TEXTLIST E_ComponentTypes
  0 = 'NA'
  10 = 'Cylinder'
  11 = 'Axis'
  20 = 'EstopButton'
  21 = 'EstopBumper'
  22 = 'Pushbutton'
  23 = 'Switch'
  30 = 'SafeIO'
  31 = 'Rio_Box'
  32 = 'Rio_Slot'
  33 = 'Encoder'
  34 = 'DiSensor'
  40 = 'ServoDrive'
  50 = 'HMI'
  51 = 'RemoteOS'
  52 = 'RemoteDB'
  60 = 'Assembly'
  61 = 'SubAssembly'
  100 = 'MainProgram'
  101 = 'StepProgram'
  102 = 'FunctionBlock'
   = ''
END_TEXTLIST

(* stored: Version 1.1.0.1, ProductVersion 3.1.4024.3
   TextList E_ComponentTypes: Id {52c6a03f-706b-4cd3-90e7-349cc2db4c63} *)
